(* Schneider Machine Expert - Basic project Lab-08-M221-delivery, file version 2.6.0.0 *)
(* ProjectInformations: Name=New project *)

HARDWARE
  Cpu 0: TM221M16R/G
  ModuleExtensionObject 0: TM3DI16K
  EthernetConfiguration: NetworkName=M221, IpAllocationMode=FixedAddress, IpAddress=0.0.0.0, SubnetMask=0.0.0.0
  SerialLineConfiguration: Baud=Baud19200, Parity=ParityEven, DataBits=DataBits8, StopBits=StopBits1, PhysicalMedium=PhysicalMediumRs485, TransmissionMode=TransmissionModeModbusRtu, SlaveId=1, Addressing=SlaveAddressing
  MastTask: UsePeriodScanMode=false, PeriodScan=100
  FastTask: Period=255
  CpuBehavior: StartingMode=StartAsPreviousState, AutoSaveRamOnEeprom=true, WatchdogPeriod=250

SYMBOLS  (address, symbol, comment, settings)
  %M0       ANYPOS
  %M1       MOVING
  %M2       DRV_EN
  %M3       DRV_FW
  %M4       DRV_RV
  %MW0      POS_BUF
  %MW1      POS_NUM
  %MW2      CALL_BUF
  %MW10     TMPBUF
  %KW0      POS_CNT  [Value=8]
  %TM0      CALL_TM  [Type=TOF, Preset=20, Base=OneHundredMilliSeconds]
  %I0.0     POS
  %Q0.0     FW
  %Q0.1     RV
  %I1.0     BTN
  %I1.8     RUN
  %I1.9     STOP

POU Generic functions
  (* SectionNumber=1 *)

// Rung 0
// Detect motion
  LD %Q0.0                (* FW *)
  OR %Q0.1                (* RV *)
  ST %M1                  (* MOVING *)
  // as ST:
  //   MOVING := FW OR RV;

// Rung 1
// Detect any position
  LD 1
  MPS
  [ %MW0 := %I0.0:8 ]     (* POS_BUF, POS *)
  MPP
  AND [ %MW0 > 0 ]        (* POS_BUF *)
  ST %M0                  (* ANYPOS *)
  // as ST:
  //   POS_BUF := POS:8;
  //   ANYPOS := POS_BUF > 0;

// Rung 2
// Detect position number: init
  LDR %M0                 (* ANYPOS *)
  [ %MW10 := %MW0 ]       (* TMPBUF, POS_BUF *)
  [ %MW1 := 0 ]           (* POS_NUM *)
  // as ST:
  //   IF RISING(ANYPOS) THEN TMPBUF := POS_BUF; END_IF;
  //   IF RISING(ANYPOS) THEN POS_NUM := 0; END_IF;

// Rung 3 %L0
// Detect position number: loop
  %L0:
  LD %M0                  (* ANYPOS *)
  AND [ %MW10 > 0 ]       (* TMPBUF *)
  [ INC %MW1 ]            (* POS_NUM *)
  [ %MW10 := SHR ( %MW10 , 1 ) ](* TMPBUF, TMPBUF *)
  JMPC %L0
  // as ST:
  //   %L0:
  //   IF ANYPOS AND TMPBUF > 0 THEN INC POS_NUM; END_IF;
  //   _t1 := ANYPOS AND TMPBUF > 0;
  //   IF _t1 THEN TMPBUF := SHR ( TMPBUF , 1 ); END_IF;
  //   IF _t1 THEN JMP %L0; END_IF;

POU Motion control
  (* SectionNumber=2 *)

// Rung 4
// Move forward/backward
  LD %M2                  (* DRV_EN *)
  MPS
  AND %M3                 (* DRV_FW *)
  ST %Q0.0                (* FW *)
  MPP
  AND %M4                 (* DRV_RV *)
  ST %Q0.1                (* RV *)
  // as ST:
  //   FW := DRV_EN AND DRV_FW;
  //   RV := DRV_EN AND DRV_RV;

// Rung 5
// Start condition
  LDR %I1.8               (* RUN *)
  MPS
  AND [ %MW1 < %KW0 ]     (* POS_NUM, POS_CNT *)
  S %M3                   (* DRV_FW *)
  MPP
  AND [ %MW1 = %KW0 ]     (* POS_NUM, POS_CNT *)
  S %M4                   (* DRV_RV *)
  // as ST:
  //   IF RISING(RUN) AND POS_NUM < POS_CNT THEN DRV_FW := TRUE; END_IF;
  //   IF RISING(RUN) AND POS_NUM = POS_CNT THEN DRV_RV := TRUE; END_IF;

// Rung 6
// Stop condition
  LDR %I1.9               (* STOP *)
  R %M3                   (* DRV_FW *)
  R %M4                   (* DRV_RV *)
  // as ST:
  //   IF RISING(STOP) THEN DRV_FW := FALSE; END_IF;
  //   IF RISING(STOP) THEN DRV_RV := FALSE; END_IF;

// Rung 7
// Reverse at edge position
  LD %M1                  (* MOVING *)
  ANDR %M0                (* ANYPOS *)
  MPS
  AND [ %MW1 = 1 ]        (* POS_NUM *)
  R %M4                   (* DRV_RV *)
  S %M3                   (* DRV_FW *)
  MPP
  AND [ %MW1 = %KW0 ]     (* POS_NUM, POS_CNT *)
  R %M3                   (* DRV_FW *)
  S %M4                   (* DRV_RV *)
  // as ST:
  //   IF MOVING AND RISING(ANYPOS) AND POS_NUM = 1 THEN DRV_RV := FALSE; END_IF;
  //   IF MOVING AND RISING(ANYPOS) AND POS_NUM = 1 THEN DRV_FW := TRUE; END_IF;
  //   IF MOVING AND RISING(ANYPOS) AND POS_NUM = POS_CNT THEN DRV_FW := FALSE; END_IF;
  //   IF MOVING AND RISING(ANYPOS) AND POS_NUM = POS_CNT THEN DRV_RV := TRUE; END_IF;

POU Call manager
  (* SectionNumber=3 *)

// Rung 8
// Call timer - stop motion
  LD %TM0.Q               (* CALL_TM *)
  STN %M2                 (* DRV_EN *)
  // as ST:
  //   DRV_EN := NOT CALL_TM.Q;

// Rung 9
// Detect any call
  LD 1
  MPS
  [ %MW10 := %I1.0:8 ]    (* TMPBUF, BTN *)
  MPP
  AND [ %MW10 > 0 ]       (* TMPBUF *)
  [ %MW2 := %MW2 OR %MW10 ](* CALL_BUF, CALL_BUF, TMPBUF *)
  [ %MW10 := 0 ]          (* TMPBUF *)
  // as ST:
  //   TMPBUF := BTN:8;
  //   IF TMPBUF > 0 THEN CALL_BUF := CALL_BUF OR TMPBUF; END_IF;
  //   IF TMPBUF > 0 THEN TMPBUF := 0; END_IF;

// Rung 10
// Process call
  LDR %M0                 (* ANYPOS *)
  MPS
  [ %MW10 := %MW2 AND %MW0 ](* TMPBUF, CALL_BUF, POS_BUF *)
  MPP
  AND [ %MW10 > 0 ]       (* TMPBUF *)
  IN %TM0                 (* CALL_TM *)
  [ %MW2 := %MW2 AND NOT ( %MW0 ) ](* CALL_BUF, CALL_BUF, POS_BUF *)
  [ %MW10 := 0 ]          (* TMPBUF *)
  // as ST:
  //   IF RISING(ANYPOS) THEN TMPBUF := CALL_BUF AND POS_BUF; END_IF;
  //   CALL_TM(IN := RISING(ANYPOS) AND TMPBUF > 0);
  //   IF RISING(ANYPOS) AND TMPBUF > 0 THEN CALL_BUF := CALL_BUF AND NOT ( POS_BUF ); END_IF;
  //   IF RISING(ANYPOS) AND TMPBUF > 0 THEN TMPBUF := 0; END_IF;
